(*
SPDX-FileCopyrightText: © 2026 Oleksandr Tiutyk <trofimich@gmail.com>
SPDX-License-Identifier: MIT
License: https://opensource.org/license/mit
*)

INTERFACE IBubbleEventDispatcher EXTENDS IObject

METHOD BubbleEvent
VAR_INPUT
	event : IEvent;
END_VAR
END_METHOD

END_INTERFACE

(* stored: Version 1.1.0.1
   Itf IBubbleEventDispatcher: Id {f62a5f0e-5516-42ac-a0e7-a8a62a6e4765}
   Method BubbleEvent: Id {acb4d73c-1a1e-40ac-a587-a8c77cde71cc} *)
